SUBAPPLICATION TokenRingPatternDemo (* TokenRing pattern demo: five-node ring (NodeA..NodeE), a real cycle rather than a two-node back-and-forth *)
  (* Standard: 61499-2; Description: Copyright (c) 2026 Meisterschulen am Ostbahnhof This program and the accompanying materials are made available under the terms of the Eclipse Public License 2.0 which is available at https://www.eclipse.org/legal/epl-2.0/ SPDX-License-Identifier: EPL-2.0 *)
  (* Version 1.1, 2026-08-31, Franz Höpfinger, Meisterschulen am Ostbahnhof, Expanded from a 2-node pair to a real 5-node ring (2 nodes is just a back-and-forth, not a ring) *)
  (* Version 1.0, 2026-08-31, Franz Höpfinger, Meisterschulen am Ostbahnhof, Mutual Exclusion / TokenRing design pattern (IEC 61499 primer course, Module 6, Valeriy Vyatkin), demo application *)
  PACKAGE Meins::DesingPatterns::TokenRingPattern;
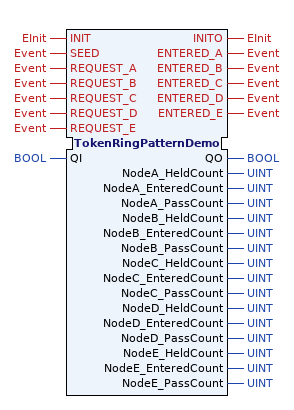
  EVENT_INPUT
    INIT : EInit; (* Initialization Request *)
    SEED; (* Bootstrap the ring: inject the token at NodeA once, after INIT *)
    REQUEST_A; (* NodeA: request the critical section for its next token hold *)
    REQUEST_B; (* NodeB: request the critical section for its next token hold *)
    REQUEST_C; (* NodeC: request the critical section for its next token hold *)
    REQUEST_D; (* NodeD: request the critical section for its next token hold *)
    REQUEST_E; (* NodeE: request the critical section for its next token hold *)
  END_EVENT
  EVENT_OUTPUT
    INITO : EInit; (* Initialization Confirm *)
    ENTERED_A; (* NodeA entered its critical section *)
    ENTERED_B; (* NodeB entered its critical section *)
    ENTERED_C; (* NodeC entered its critical section *)
    ENTERED_D; (* NodeD entered its critical section *)
    ENTERED_E; (* NodeE entered its critical section *)
  END_EVENT
  VAR_INPUT
    QI : BOOL; (* Input event qualifier *)
  END_VAR
  VAR_OUTPUT
    QO : BOOL; (* Output event qualifier *)
    NodeA_HeldCount : UINT; (* NodeA: number of times it received the token *)
    NodeA_EnteredCount : UINT; (* NodeA: number of times it used the critical section *)
    NodeA_PassCount : UINT; (* NodeA: number of acknowledged hand-offs *)
    NodeB_HeldCount : UINT; (* NodeB: number of times it received the token *)
    NodeB_EnteredCount : UINT; (* NodeB: number of times it used the critical section *)
    NodeB_PassCount : UINT; (* NodeB: number of acknowledged hand-offs *)
    NodeC_HeldCount : UINT; (* NodeC: number of times it received the token *)
    NodeC_EnteredCount : UINT; (* NodeC: number of times it used the critical section *)
    NodeC_PassCount : UINT; (* NodeC: number of acknowledged hand-offs *)
    NodeD_HeldCount : UINT; (* NodeD: number of times it received the token *)
    NodeD_EnteredCount : UINT; (* NodeD: number of times it used the critical section *)
    NodeD_PassCount : UINT; (* NodeD: number of acknowledged hand-offs *)
    NodeE_HeldCount : UINT; (* NodeE: number of times it received the token *)
    NodeE_EnteredCount : UINT; (* NodeE: number of times it used the critical section *)
    NodeE_PassCount : UINT; (* NodeE: number of acknowledged hand-offs *)
  END_VAR
  FBS
    NodeA : Meins::DesingPatterns::TokenRingPattern::TokenRingNode;
    NodeB : Meins::DesingPatterns::TokenRingPattern::TokenRingNode;
    NodeC : Meins::DesingPatterns::TokenRingPattern::TokenRingNode;
    NodeD : Meins::DesingPatterns::TokenRingPattern::TokenRingNode;
    NodeE : Meins::DesingPatterns::TokenRingPattern::TokenRingNode;
  END_FBS
  EVENT_CONNECTIONS
    INIT TO NodeA.INIT;
    NodeA.INITO TO NodeB.INIT;
    NodeB.INITO TO NodeC.INIT;
    NodeC.INITO TO NodeD.INIT;
    NodeD.INITO TO NodeE.INIT;
    NodeE.INITO TO INITO;
    SEED TO NodeA.SEED;
    REQUEST_A TO NodeA.REQUEST;
    REQUEST_B TO NodeB.REQUEST;
    REQUEST_C TO NodeC.REQUEST;
    REQUEST_D TO NodeD.REQUEST;
    REQUEST_E TO NodeE.REQUEST;
    NodeA.ENTERED TO ENTERED_A;
    NodeB.ENTERED TO ENTERED_B;
    NodeC.ENTERED TO ENTERED_C;
    NodeD.ENTERED TO ENTERED_D;
    NodeE.ENTERED TO ENTERED_E;
  END_CONNECTIONS
  DATA_CONNECTIONS
    QI TO NodeA.QI;
    NodeA.QO TO NodeB.QI;
    NodeB.QO TO NodeC.QI;
    NodeC.QO TO NodeD.QI;
    NodeD.QO TO NodeE.QI;
    NodeE.QO TO QO;
    NodeA.HeldCount TO NodeA_HeldCount;
    NodeA.EnteredCount TO NodeA_EnteredCount;
    NodeA.PassCount TO NodeA_PassCount;
    NodeB.HeldCount TO NodeB_HeldCount;
    NodeB.EnteredCount TO NodeB_EnteredCount;
    NodeB.PassCount TO NodeB_PassCount;
    NodeC.HeldCount TO NodeC_HeldCount;
    NodeC.EnteredCount TO NodeC_EnteredCount;
    NodeC.PassCount TO NodeC_PassCount;
    NodeD.HeldCount TO NodeD_HeldCount;
    NodeD.EnteredCount TO NodeD_EnteredCount;
    NodeD.PassCount TO NodeD_PassCount;
    NodeE.HeldCount TO NodeE_HeldCount;
    NodeE.EnteredCount TO NodeE_EnteredCount;
    NodeE.PassCount TO NodeE_PassCount;
  END_CONNECTIONS
  ADAPTER_CONNECTIONS
    NodeA.MTXOUT TO NodeB.MTXIN; (* NodeA gives the token to NodeB *)
    NodeB.MTXOUT TO NodeC.MTXIN; (* NodeB gives the token to NodeC *)
    NodeC.MTXOUT TO NodeD.MTXIN; (* NodeC gives the token to NodeD *)
    NodeD.MTXOUT TO NodeE.MTXIN; (* NodeD gives the token to NodeE *)
    NodeE.MTXOUT TO NodeA.MTXIN; (* NodeE gives the token back to NodeA, closing the ring *)
  END_CONNECTIONS
END_SUBAPPLICATION
